(* IEC 61131-3 sources: Industry-PLC-LLM/data/PLCBEAD_repo/PLCBEAD_PLCEmbed-main/PLC-BEAD/Source/GEB/SHR_4E, 1 file *)

(* ---- SHR_4E.ST ---- *)
FUNCTION_BLOCK SHR_4E_Block

	VAR_INPUT
		SET :	BOOL;
		D0 :	BOOL;
		CLK :	BOOL;
		RST :	BOOL;
	END_VAR

	VAR_OUTPUT
		Q0 :	BOOL;
		Q1 :	BOOL;
		Q2 :	BOOL;
		Q3 :	BOOL;
	END_VAR

	VAR
		TRIG :	R_TRIG;
	END_VAR

	TRIG(CLK := CLK);

	IF SET OR RST THEN
		Q0 := NOT RST;
		Q1 := Q0;
		Q2 := Q0;
		Q3 := Q0;
	ELSIF TRIG.Q THEN
		Q3 := Q2;
		Q2 := Q1;
		Q1 := Q0;
		Q0 := D0;
	END_IF;

END_FUNCTION_BLOCK

PROGRAM program0

	VAR
		SET :	BOOL;
		D0 :	BOOL;
		CLK :	BOOL;
		RST :	BOOL;
		Q0 :	BOOL;
		Q1 :	BOOL;
		Q2 :	BOOL;
		Q3 :	BOOL;
		func_block : SHR_4E_Block;
	END_VAR
	func_block.SET  :=SET;
	func_block.D0  :=D0;
	func_block.CLK  :=CLK;
	func_block.RST  :=RST;
	func_block();
	Q0 := func_block.Q0;
	Q1 := func_block.Q1;
	Q2 := func_block.Q2;
	Q3 := func_block.Q3;

END_PROGRAM
